FUNCTION EtaHasBit : BOOL
VAR_INPUT
	w		: WORD;
	bBit	: INT;
END_VAR

EtaHasBit := (w AND SHL(WORD#1, bBit)) <> 0;

END_FUNCTION

(* stored: Version 1.1.0.1, ProductVersion 3.1.4024.15
   POU EtaHasBit: Id {170bfd13-bf01-491b-96d8-8ba34effd3c7}, SpecialFunc None *)
